FUNCTION_BLOCK RequestConsumer
  (* Standard: 61499-2 *)
  (* Version 0.1, 2014-00-16, Canto-Air, CANTO-AIR-PC *)
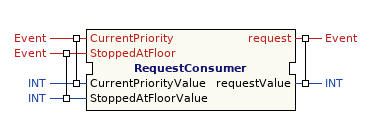
  EVENT_INPUT
    CurrentPriority WITH CurrentPriorityValue;
    StoppedAtFloor WITH StoppedAtFloorValue;
  END_EVENT
  EVENT_OUTPUT
    request WITH requestValue;
  END_EVENT
  VAR_INPUT
    CurrentPriorityValue : INT;
    StoppedAtFloorValue : INT;
  END_VAR
  VAR_OUTPUT
    requestValue : INT;
  END_VAR
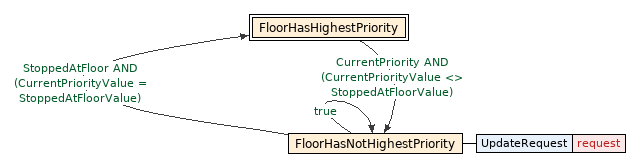
  EC_STATES
    FloorHasHighestPriority;
    FloorHasNotHighestPriority : UpdateRequest -> request;
  END_STATES
  EC_TRANSITIONS
    FloorHasHighestPriority TO FloorHasNotHighestPriority := CurrentPriority AND (CurrentPriorityValue <> StoppedAtFloorValue);
    FloorHasNotHighestPriority TO FloorHasHighestPriority := StoppedAtFloor AND (CurrentPriorityValue = StoppedAtFloorValue);
    FloorHasNotHighestPriority TO FloorHasNotHighestPriority := true;
  END_TRANSITIONS
  ALGORITHM UpdateRequest IN C:
me->requestValue = me->CurrentPriorityValue;
  END_ALGORITHM
END_FUNCTION_BLOCK
